TEXTLIST PXExitYesNo
  FALSE = 'NO'
  TRUE = 'YES'
   = ''
END_TEXTLIST

(* stored: Version 1.1.0.1, ProductVersion 3.1.4024.11
   TextList PXExitYesNo: Id {348910f5-8ee5-46e0-9258-e0f09a9fa6f7} *)
